(* PLC project  *)

TYPE MyEnum : (Value1, Value2, Value3);
END_TYPE

TYPE MyArray : ARRAY[0..9] OF LINT;
END_TYPE

TYPE MyStruct : STRUCT
  Field1 : BOOL;
  Field2 : LREAL;
  Field3 : TIME;
  Field4 : DATE;
  Field5 : MyEnum;
END_STRUCT;
END_TYPE

TYPE MySubrange : INT(-100..100);
END_TYPE
